FUNCTION_BLOCK SUBSCRIBE_21 (* Six-variable Subscriber *)
  (* Standard: 61499-2 *)
  (* Version 0.0, 2004-06-09, JHC, Rockwell Automation, Derived from SUBSCRIBE_4. *)
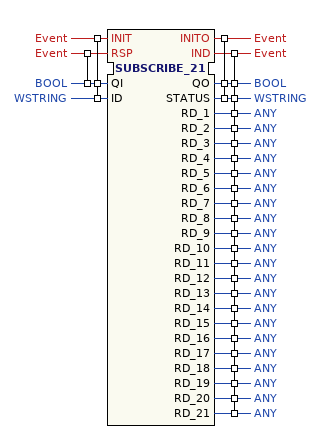
  EVENT_INPUT
    INIT WITH QI, ID; (* Service Initialization *)
    RSP WITH QI; (* Service Response *)
  END_EVENT
  EVENT_OUTPUT
    INITO WITH QO, STATUS; (* Initialization Confirm *)
    IND WITH QO, STATUS, RD_1, RD_2, RD_3, RD_4, RD_5, RD_6, RD_7, RD_8, RD_9, RD_10, RD_11, RD_12, RD_13, RD_14, RD_15, RD_16, RD_17, RD_18, RD_19, RD_20, RD_21; (* Service Indication *)
  END_EVENT
  VAR_INPUT
    QI : BOOL; (* Event Input Qualifier *)
    ID : WSTRING; (* Connection Identifier *)
  END_VAR
  VAR_OUTPUT
    QO : BOOL; (* Event Output Qualifier *)
    STATUS : WSTRING; (* Service Status *)
    RD_1 : ANY; (* Subscribed Data *)
    RD_2 : ANY; (* Subscribed Data *)
    RD_3 : ANY; (* Subscribed Data *)
    RD_4 : ANY; (* Subscribed Data *)
    RD_5 : ANY; (* Subscribed Data *)
    RD_6 : ANY; (* Subscribed Data *)
    RD_7 : ANY; (* Subscribed Data *)
    RD_8 : ANY; (* Subscribed Data *)
    RD_9 : ANY; (* Subscribed Data *)
    RD_10 : ANY; (* Subscribed Data *)
    RD_11 : ANY; (* Subscribed Data *)
    RD_12 : ANY; (* Subscribed Data *)
    RD_13 : ANY; (* Subscribed Data *)
    RD_14 : ANY; (* Subscribed Data *)
    RD_15 : ANY; (* Subscribed Data *)
    RD_16 : ANY; (* Subscribed Data *)
    RD_17 : ANY; (* Subscribed Data *)
    RD_18 : ANY; (* Subscribed Data *)
    RD_19 : ANY; (* Subscribed Data *)
    RD_20 : ANY; (* Subscribed Data *)
    RD_21 : ANY; (* Subscribed Data *)
  END_VAR
END_FUNCTION_BLOCK
